// TIA Portal V19 export
FUNCTION "FC_004_ModularConvoyers" : Void   // FC11, LAD
{ S7_Optimized_Access := 'TRUE' }
// stored: SetENOAutomatically false
BEGIN

REGION Network 1 (SCL)
   //************************************************************
   //===Author: Mateusz Połojko
   //-----Linkedin: https://pl.linkedin.com/in/mateusz-po%C5%82ojko-52a3541b1
   //-----Github: https://github.com/Bhazel95
   //===Description:
   //-----Control of the transporter and executive modules
   //===Customer:
   //-----Apator Powogaz S.A.
   //************************************************************
END_REGION

REGION Network 2
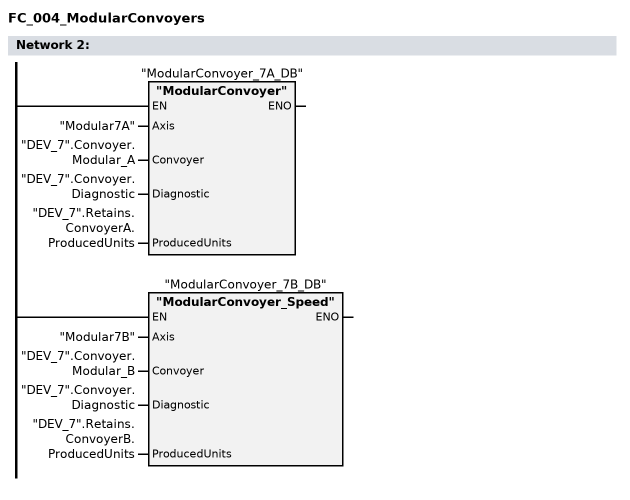
   RUNG wire#powerrail
      "ModularConvoyer_7A_DB"(Axis := "Modular7A", Convoyer := "DEV_7".Convoyer.Modular_A, Diagnostic := "DEV_7".Convoyer.Diagnostic, ProducedUnits := "DEV_7".Retains.ConvoyerA.ProducedUnits)
   END_RUNG
   RUNG wire#powerrail
      "ModularConvoyer_7B_DB"(Axis := "Modular7B", Convoyer := "DEV_7".Convoyer.Modular_B, Diagnostic := "DEV_7".Convoyer.Diagnostic, ProducedUnits := "DEV_7".Retains.ConvoyerB.ProducedUnits)
   END_RUNG
   // the same network as SCL:
   "ModularConvoyer_7A_DB"(Axis := "Modular7A",   // "ModularConvoyer"
                           Convoyer := "DEV_7".Convoyer.Modular_A,
                           Diagnostic := "DEV_7".Convoyer.Diagnostic,
                           ProducedUnits := "DEV_7".Retains.ConvoyerA.ProducedUnits);
   "ModularConvoyer_7B_DB"(Axis := "Modular7B",   // "ModularConvoyer_Speed"
                           Convoyer := "DEV_7".Convoyer.Modular_B,
                           Diagnostic := "DEV_7".Convoyer.Diagnostic,
                           ProducedUnits := "DEV_7".Retains.ConvoyerB.ProducedUnits);
END_REGION
END_FUNCTION
